// TIA Portal V16 export
// export: Created 2024-09-05T17:39:16.3052633Z, ExportSetting WithDefaults, DisplayName Totally Integrated Automation Portal, DisplayVersion V16 Update 6, DisplayName TIA Portal Version Control Interface, DisplayVersion V16 Update 2, DisplayName TIA Portal Openness, DisplayVersion V16 Update 6, DisplayName STEP 7 Professional, DisplayVersion V16 Update 6, DisplayName STEP 7 Safety, DisplayVersion V16, DisplayName WinCC Advanced, DisplayVersion V16 Update 6
FUNCTION "FC_ProductionProgram" : Void   // FC6100, LAD
{ S7_Optimized_Access := 'TRUE' }
VERSION : 0.1
// stored: AutoNumber false, IsIECCheckEnabled false, SetENOAutomatically false, UDAEnableTagReadback false
   VAR_INPUT
      iSettingsSecurity : Bool;
      iBlinker : Bool;
   END_VAR
BEGIN

REGION Network 1 (SCL): Production program edit
   //Actual program
   IF "DB_ProductionProgramActual".ProgrammNumber < 1 OR "DB_ProductionProgramActual".ProgrammNumber > "NumberOfProductionPrograms" THEN
       "DB_ProductionProgramActual".ProgrammNumber := 1;
   END_IF;
   "DB_ProductionProgramActual".Program := "DB_ProductionProgramList".Program["DB_ProductionProgramActual".ProgrammNumber];
   "DB_ProductionProgramActual".Program.CupformingParametersRight.ApproachForce := "DB_ProductionProgramActual".Program.CupformingParametersLeft.ApproachForce;
   "DB_ProductionProgramActual".Program.CupformingParametersRight.FinalForce := "DB_ProductionProgramActual".Program.CupformingParametersLeft.FinalForce;

   //Program to edit: Number limits
   IF "DB_ProductionProgramEdit".Commands.ProgramEdit.Number < 1 THEN
       "DB_ProductionProgramEdit".Commands.ProgramEdit.Number := 1;
   END_IF;

   IF "DB_ProductionProgramEdit".Commands.ProgramEdit.Number > "NumberOfProductionPrograms" THEN
       "DB_ProductionProgramEdit".Commands.ProgramEdit.Number := "NumberOfProductionPrograms";
   END_IF;

   //Program to edit: Number changed
   "DB_ProductionProgramEdit".Commands.ProgramEdit.NumberChanged := FALSE;
   IF "DB_ProductionProgramEdit".Commands.ProgramEdit.Number <> "DB_ProductionProgramEdit".Commands.ProgramEdit.NumberLast THEN
       "DB_ProductionProgramEdit".Commands.ProgramEdit.NumberLast := "DB_ProductionProgramEdit".Commands.ProgramEdit.Number;
       "DB_ProductionProgramEdit".Commands.ProgramEdit.NumberChanged := TRUE;
   END_IF;

   //Program to edit: Load
   IF #iSettingsSecurity = FALSE OR
       "DB_ProductionProgramEdit".Commands.ProgramEdit.NumberChanged = TRUE OR
       "DB_ProductionProgramEdit".Commands.ProgramEdit.LoadAll = TRUE THEN
       "DB_ProductionProgramEdit".Commands.ProgramEdit.Commands := 1;
   END_IF;

   IF "DB_ProductionProgramEdit".Commands.ProgramEdit.Commands = 1 THEN
       "DB_ProductionProgramEdit".ProgramEdit := "DB_ProductionProgramList".Program["DB_ProductionProgramEdit".Commands.ProgramEdit.Number];
       "READER_MODEL_ACTUAL".EDIT := "READER_MODEL".PRODUCT["DB_ProductionProgramEdit".Commands.ProgramEdit.Number];
   END_IF;

   //Product to edit: Number limits
   IF "DB_ProductionProgramEdit".Commands.ProgramEdit.NumberChanged = TRUE OR
       "DB_ProductionProgramEdit".Commands.ProgramEdit.LoadAll = TRUE THEN
       "DB_ProductionProgramEdit".Commands.ProductEdit.Number := 1;
   END_IF;

   IF "DB_ProductionProgramEdit".Commands.ProductEdit.Number < 1 THEN
       "DB_ProductionProgramEdit".Commands.ProductEdit.Number := 1;
   END_IF;

   IF "DB_ProductionProgramEdit".Commands.ProductEdit.Number > "NumberOfProductionProducts" THEN
       "DB_ProductionProgramEdit".Commands.ProductEdit.Number := "NumberOfProductionProducts";
   END_IF;

   //Product to edit: Number changed
   "DB_ProductionProgramEdit".Commands.ProductEdit.NumberChanged := FALSE;
   IF "DB_ProductionProgramEdit".Commands.ProductEdit.Number <> "DB_ProductionProgramEdit".Commands.ProductEdit.NumberLast THEN
       "DB_ProductionProgramEdit".Commands.ProductEdit.NumberLast := "DB_ProductionProgramEdit".Commands.ProductEdit.Number;
       "DB_ProductionProgramEdit".Commands.ProductEdit.NumberChanged := TRUE;
   END_IF;


   //Position to edit: Number limits
   IF "DB_ProductionProgramEdit".Commands.ProgramEdit.NumberChanged = TRUE OR
       "DB_ProductionProgramEdit".Commands.ProgramEdit.LoadAll = TRUE OR
       "DB_ProductionProgramEdit".Commands.ProductEdit.NumberChanged = TRUE THEN
       "DB_ProductionProgramEdit".Commands.PositionEdit.Number := 1;
   END_IF;

   IF "DB_ProductionProgramEdit".Commands.PositionEdit.Number < 1 THEN
       "DB_ProductionProgramEdit".Commands.PositionEdit.Number := 1;
   END_IF;

   //Position to edit: Number changed
   "DB_ProductionProgramEdit".Commands.PositionEdit.NumberChanged := FALSE;
   IF "DB_ProductionProgramEdit".Commands.PositionEdit.Number <> "DB_ProductionProgramEdit".Commands.PositionEdit.NumberLast THEN
       "DB_ProductionProgramEdit".Commands.PositionEdit.NumberLast := "DB_ProductionProgramEdit".Commands.PositionEdit.Number;
       "DB_ProductionProgramEdit".Commands.PositionEdit.NumberChanged := TRUE;
   END_IF;

   //Position to edit: Load
   "DB_ProductionProgramEdit".Commands.PositionEdit.Load := FALSE;
   IF "DB_ProductionProgramEdit".Commands.ProgramEdit.Commands = 1 OR
       "DB_ProductionProgramEdit".Commands.ProductEdit.NumberChanged = TRUE OR
       "DB_ProductionProgramEdit".Commands.PositionEdit.NumberChanged = TRUE THEN
       "DB_ProductionProgramEdit".Commands.PositionEdit.Load := TRUE;
   END_IF;

   //Save program
   IF "DB_ProductionProgramEdit".Commands.ProgramEdit.Commands = 2 THEN
       "DB_ProductionProgramList".Program["DB_ProductionProgramEdit".Commands.ProgramEdit.Number] := "DB_ProductionProgramEdit".ProgramEdit;
       "READER_MODEL".PRODUCT["DB_ProductionProgramEdit".Commands.ProgramEdit.Number] :="READER_MODEL_ACTUAL".EDIT;
   END_IF;

   //Copy program
   IF "DB_ProductionProgramEdit".Commands.ProgramEdit.Commands = 3 THEN
       "DB_ProductionProgramEdit".ProgramInBox := "DB_ProductionProgramEdit".ProgramEdit;
       "DB_ProductionProgramEdit".Commands.ProgramEdit.NumberInBox := "DB_ProductionProgramEdit".Commands.ProgramEdit.Number;
       "READER_MODEL_ACTUAL".IN_BOX := "READER_MODEL_ACTUAL".EDIT;
   END_IF;

   //Paste program
   IF "DB_ProductionProgramEdit".Commands.ProgramEdit.Commands = 4 THEN
       "DB_ProductionProgramEdit".ProgramEdit := "DB_ProductionProgramEdit".ProgramInBox;
       "READER_MODEL_ACTUAL".EDIT := "READER_MODEL_ACTUAL".IN_BOX;
   END_IF;

   //Delete program
   IF "DB_ProductionProgramEdit".Commands.ProgramEdit.Commands = 5 THEN
       "DB_ProductionProgramEdit".ProgramEdit := "DB_ProductionProgramEdit".ProgramEmpty;
   END_IF;

   //Program to edit: Check if it was changed
   "DB_ProductionProgramEdit".Commands.ProgramEdit.ProgramChanged := FALSE;
   IF "DB_ProductionProgramEdit".ProgramEdit <> "DB_ProductionProgramList".Program["DB_ProductionProgramEdit".Commands.ProgramEdit.Number] OR
       "READER_MODEL_ACTUAL".EDIT <> "READER_MODEL".PRODUCT["DB_ProductionProgramEdit".Commands.ProgramEdit.Number]
   THEN
       "DB_ProductionProgramEdit".Commands.ProgramEdit.ProgramChanged := TRUE;
   END_IF;
END_REGION

REGION Network 2: Command status
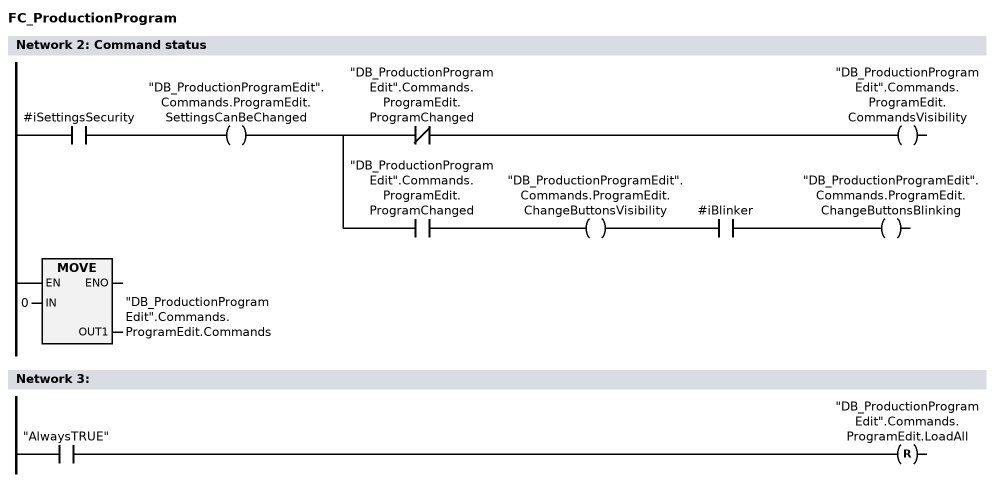
   RUNG wire#powerrail
      Contact( #iSettingsSecurity )
      Coil( "DB_ProductionProgramEdit".Commands.ProgramEdit.SettingsCanBeChanged )
      wire#w1
      I_Contact( "DB_ProductionProgramEdit".Commands.ProgramEdit.ProgramChanged )
      Coil( "DB_ProductionProgramEdit".Commands.ProgramEdit.CommandsVisibility )
   END_RUNG
   RUNG wire#w1
      Contact( "DB_ProductionProgramEdit".Commands.ProgramEdit.ProgramChanged )
      Coil( "DB_ProductionProgramEdit".Commands.ProgramEdit.ChangeButtonsVisibility )
      Contact( #iBlinker )
      Coil( "DB_ProductionProgramEdit".Commands.ProgramEdit.ChangeButtonsBlinking )
   END_RUNG
   RUNG wire#powerrail
      Move(in := 0, out1 => "DB_ProductionProgramEdit".Commands.ProgramEdit.Commands)
   END_RUNG
   // the same network as SCL:
   "DB_ProductionProgramEdit".Commands.ProgramEdit.SettingsCanBeChanged := #iSettingsSecurity;
   "DB_ProductionProgramEdit".Commands.ProgramEdit.CommandsVisibility := #iSettingsSecurity AND NOT "DB_ProductionProgramEdit".Commands.ProgramEdit.ProgramChanged;
   "DB_ProductionProgramEdit".Commands.ProgramEdit.ChangeButtonsVisibility := #iSettingsSecurity AND "DB_ProductionProgramEdit".Commands.ProgramEdit.ProgramChanged;
   "DB_ProductionProgramEdit".Commands.ProgramEdit.ChangeButtonsBlinking := "DB_ProductionProgramEdit".Commands.ProgramEdit.ChangeButtonsVisibility AND #iBlinker;
   "DB_ProductionProgramEdit".Commands.ProgramEdit.Commands := 0;
END_REGION

REGION Network 3
   RUNG wire#powerrail
      Contact( "AlwaysTRUE" )
      R_Coil( "DB_ProductionProgramEdit".Commands.ProgramEdit.LoadAll )
   END_RUNG
   // the same network as SCL:
   IF "AlwaysTRUE" THEN "DB_ProductionProgramEdit".Commands.ProgramEdit.LoadAll := FALSE; END_IF;
END_REGION
END_FUNCTION
